// Mitsubishi GX Works2 project: BookEX6_33 Bit   PLC: Q13UDV

// global labels: Global
VAR_GLOBAL
  bVar0 AT M5000 : BOOL;
  abArray0 AT M5010 : ARRAY [0..49] OF BOOL;
  sStr0 AT D5000 : STRING[199];
  sStr1 AT D5100 : STRING[199];
  sStr2 AT D5200 : STRING[199];
  sStr3 AT D5300 : STRING[199];
  sStr4 AT D5400 : STRING[199];
  sStr5 AT D5500 : STRING[199];
  sStr6 AT D5600 : STRING[199];
  sStr7 AT D5700 : STRING[199];
  sStr8 AT D5800 : STRING[199];
  sStr9 AT D5900 : STRING[199];
  iVar0 AT D4500 : INT;
  iVar1 AT D4501 : INT;
  iVar2 AT D4502 : INT;
  iVar3 AT D4503 : INT;
  iVar4 AT D4504 : INT;
  iVar5 AT D4505 : INT;
  iVar6 AT D4506 : INT;
  iVar7 AT D4507 : INT;
  iVar8 AT D4508 : INT;
  iVar9 AT D4509 : INT;
  dVar0 AT D4510 : DINT;
  dVar1 AT D4512 : DINT;
  dVar2 AT D4514 : DINT;
  dVar3 AT D4516 : DINT;
  dVar4 AT D4518 : DINT;
  dVar5 AT D4520 : DINT;
  dVar6 AT D4522 : DINT;
  dVar7 AT D4524 : DINT;
  dVar8 AT D4526 : DINT;
  dVar9 AT D4528 : DINT;
  wVar0 AT D4530 : WORD;
  wVar1 AT D4531 : WORD;
  wVar2 AT D4532 : WORD;
  wVar3 AT D4533 : WORD;
  wVar4 AT D4534 : WORD;
  wVar5 AT D4535 : WORD;
  wVar6 AT D4536 : WORD;
  wVar7 AT D4537 : WORD;
  wVar8 AT D4538 : WORD;
  wVar9 AT D4539 : WORD;
  dwVar0 AT D4540 : DWORD;
  dwVar1 AT D4542 : DWORD;
  dwVar2 AT D4544 : DWORD;
  dwVar3 AT D4546 : DWORD;
  dwVar4 AT D4548 : DWORD;
  dwVar5 AT D4550 : DWORD;
  dwVar6 AT D4552 : DWORD;
  dwVar7 AT D4554 : DWORD;
  dwVar8 AT D4556 : DWORD;
  dwVar9 AT D4558 : DWORD;
  fsVar0 AT D4560 : REAL;
  fsVar1 AT D4562 : REAL;
  fsVar2 AT D4564 : REAL;
  fsVar3 AT D4566 : REAL;
  fsVar4 AT D4568 : REAL;
  fsVar5 AT D4570 : REAL;
  fsVar6 AT D4572 : REAL;
  fsVar7 AT D4574 : REAL;
  fsVar8 AT D4576 : REAL;
  fsVar9 AT D4578 : REAL;
  fdVar0 AT D4580 : LREAL;
  tTime0 AT D4620 : TIME;
  tTime1 AT D4622 : TIME;
  tTime2 AT D4624 : TIME;
  tTime3 AT D4626 : TIME;
  tTime4 AT D4628 : TIME;
  tTime5 AT D4630 : TIME;
  tTime6 AT D4632 : TIME;
  tTime7 AT D4634 : TIME;
  tTime8 AT D4636 : TIME;
  tTime9 AT D4638 : TIME;
  tTime10 AT D4640 : TIME;
  bVar1 AT M5001 : BOOL;
  bVar2 AT M5002 : BOOL;
  bVar3 AT M5003 : BOOL;
  bVar4 AT M5004 : BOOL;
  bVar5 AT M5005 : BOOL;
  bVar6 AT M5006 : BOOL;
  bVar7 AT M5007 : BOOL;
  bVar8 AT M5008 : BOOL;
  bVar9 AT M5009 : BOOL;
  abArray1 AT M5060 : ARRAY [0..49] OF BOOL;
  abArray2 AT M5110 : ARRAY [0..49] OF BOOL;
  abArray3 AT M5160 : ARRAY [0..49] OF BOOL;
  abArray4 AT M5210 : ARRAY [0..49] OF BOOL;
  abArray5 AT M5260 : ARRAY [0..49] OF BOOL;
  abArray6 AT M5310 : ARRAY [0..49] OF BOOL;
  abArray7 AT M5360 : ARRAY [0..49] OF BOOL;
  abArray8 AT M5410 : ARRAY [0..49] OF BOOL;
  abArray9 AT M5460 : ARRAY [0..49] OF BOOL;
  fdVar1 AT D4584 : LREAL;
  fdVar2 AT D4588 : LREAL;
  fdVar3 AT D4592 : LREAL;
  fdVar4 AT D4596 : LREAL;
  fdVar5 AT D4600 : LREAL;
  fdVar6 AT D4604 : LREAL;
  fdVar7 AT D4608 : LREAL;
  fdVar8 AT D4612 : LREAL;
  fdVar9 AT D4616 : LREAL;
  afsPen0 AT D2000 : ARRAY [0..499] OF REAL;
  afsPen1 AT D3000 : ARRAY [0..499] OF REAL;
END_VAR
// user libraries (not included): HMI

FUNCTION DBRST
VAR_INPUT
  dw_IN : DWORD;
  i_Pos : INT;
END_VAR
VAR
  dwInput : DWORD;
  dwTmp1 : DWORD;
  dwTmp2 : DWORD;
END_VAR
;
dwTmp1 := H00000001;
dwInput := dw_IN;
DROL(TRUE, i_Pos MOD 32, dwTmp1);
dwTmp2 := dwInput AND NOT dwTmp1;
DBRST := dwTmp2;
END_FUNCTION

FUNCTION DBSET
VAR_INPUT
  dw_IN : DWORD;
END_VAR
VAR
  dwInput : DWORD;
END_VAR
VAR_INPUT
  i_Pos : INT;
END_VAR
VAR
  dwTmp1 : DWORD;
  dwTmp2 : DWORD;
END_VAR
;
dwTmp1 := H00000001;
dwInput := dw_IN;
DROL(TRUE, i_Pos MOD 32, dwTmp1);
dwTmp2 := dwInput OR dwTmp1;
DBSET := dwTmp2;
END_FUNCTION

FUNCTION newDTEST
VAR_INPUT
  dw_IN : DWORD;
  i_Pos : INT;
END_VAR
VAR
  dwInput : DWORD;
  dwTmp1 : DWORD;
  dwTmp2 : DWORD;
END_VAR
;
dwTmp1 := H00000001;
dwInput := dw_IN;
DROL(TRUE, i_Pos MOD 32, dwTmp1);
dwTmp2 := dwInput AND dwTmp1;
newDTEST := dwTmp2 = dwTmp1;
END_FUNCTION

PROGRAM ExBKRST
(* structured ladder/FBD written out as ST: instructions are called as NAME(EN, inputs, outputs); _pN, _eN, _tN stand for wires *)
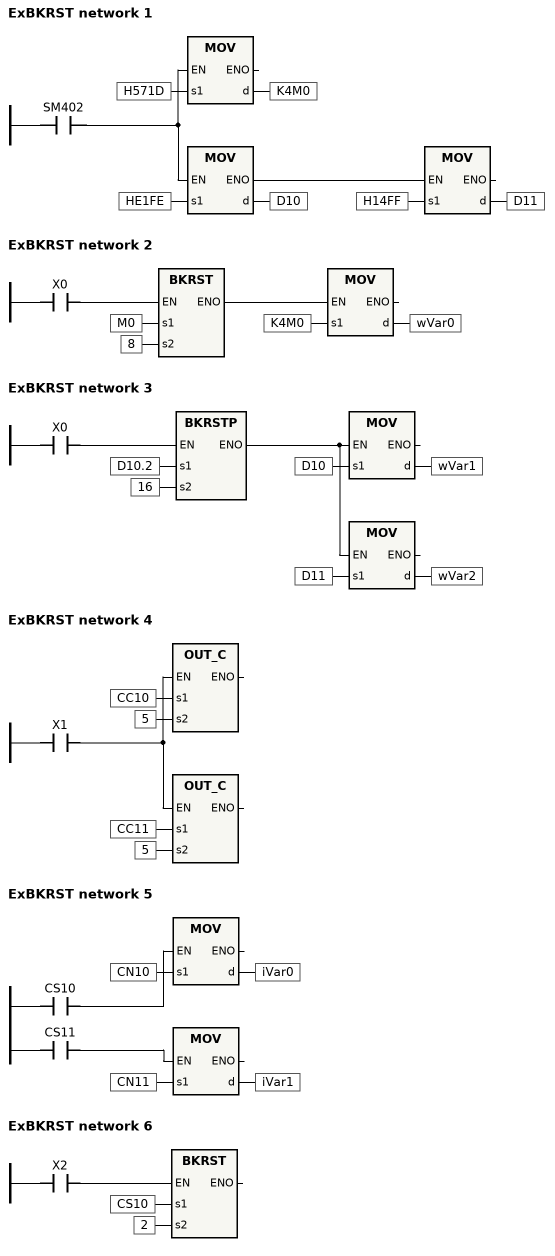
(* network 1 *)
MOV(SM402, H571D, K4M0);
_e1 := MOV(SM402, HE1FE, D10);
MOV(_e1, H14FF, D11);
(* network 2 *)
_e1 := BKRST(X0, M0, 8);
MOV(_e1, K4M0, wVar0);
(* network 3 *)
_e1 := BKRSTP(X0, D10.2, 16);
MOV(_e1, D10, wVar1);
MOV(_e1, D11, wVar2);
(* network 4 *)
OUT_C(X1, CC10, 5);
OUT_C(X1, CC11, 5);
(* network 5 *)
MOV(CS10, CN10, iVar0);
MOV(CS11, CN11, iVar1);
(* network 6 *)
BKRST(X2, CS10, 2);
END_PROGRAM

PROGRAM ExBSET
(* structured ladder/FBD written out as ST: instructions are called as NAME(EN, inputs, outputs); _pN, _eN, _tN stand for wires *)
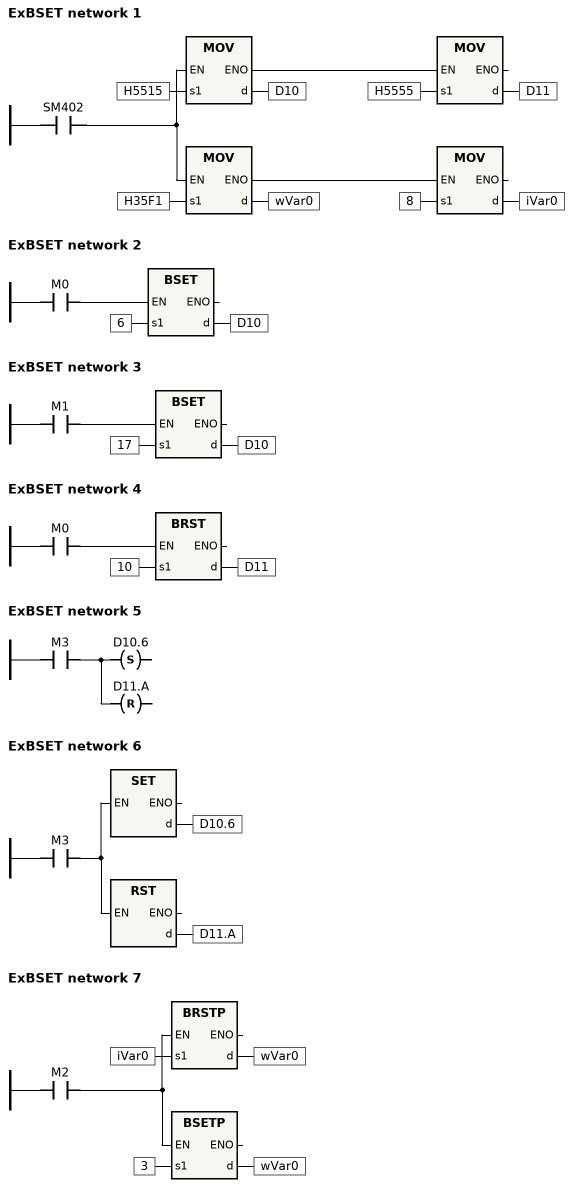
(* network 1 *)
_e1 := MOV(SM402, H5515, D10);
MOV(_e1, H5555, D11);
_e2 := MOV(SM402, H35F1, wVar0);
MOV(_e2, 8, iVar0);
(* network 2 *)
BSET(M0, 6, D10);
(* network 3 *)
BSET(M1, 17, D10);
(* network 4 *)
BRST(M0, 10, D11);
(* network 5 *)
SET(M3, D10.6);
RST(M3, D11.A);
(* network 6 *)
SET(M3, D10.6);
RST(M3, D11.A);
(* network 7 *)
BRSTP(M2, iVar0, wVar0);
BSETP(M2, 3, wVar0);
END_PROGRAM

PROGRAM ExLib
(* structured ladder/FBD written out as ST: instructions are called as NAME(EN, inputs, outputs); _pN, _eN, _tN stand for wires *)
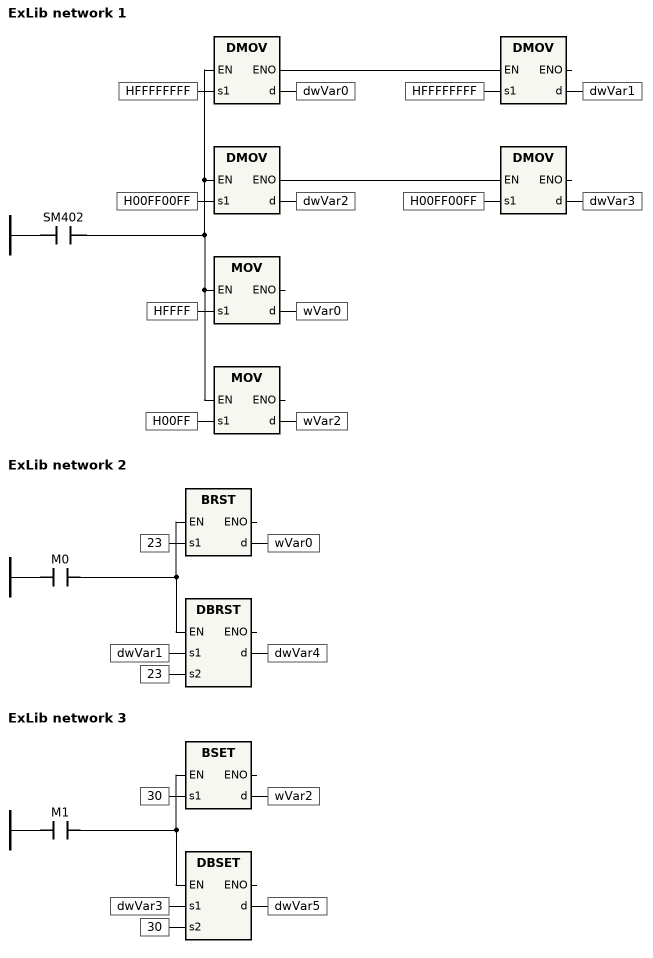
(* network 1 *)
_e1 := DMOV(SM402, HFFFFFFFF, dwVar0);
DMOV(_e1, HFFFFFFFF, dwVar1);
_e2 := DMOV(SM402, H00FF00FF, dwVar2);
DMOV(_e2, H00FF00FF, dwVar3);
MOV(SM402, HFFFF, wVar0);
MOV(SM402, H00FF, wVar2);
(* network 2 *)
BRST(M0, 23, wVar0);
DBRST(M0, dwVar1, 23, dwVar4);
(* network 3 *)
BSET(M1, 30, wVar2);
DBSET(M1, dwVar3, 30, dwVar5);
END_PROGRAM

PROGRAM ExTEST
(* structured ladder/FBD written out as ST: instructions are called as NAME(EN, inputs, outputs); _pN, _eN, _tN stand for wires *)
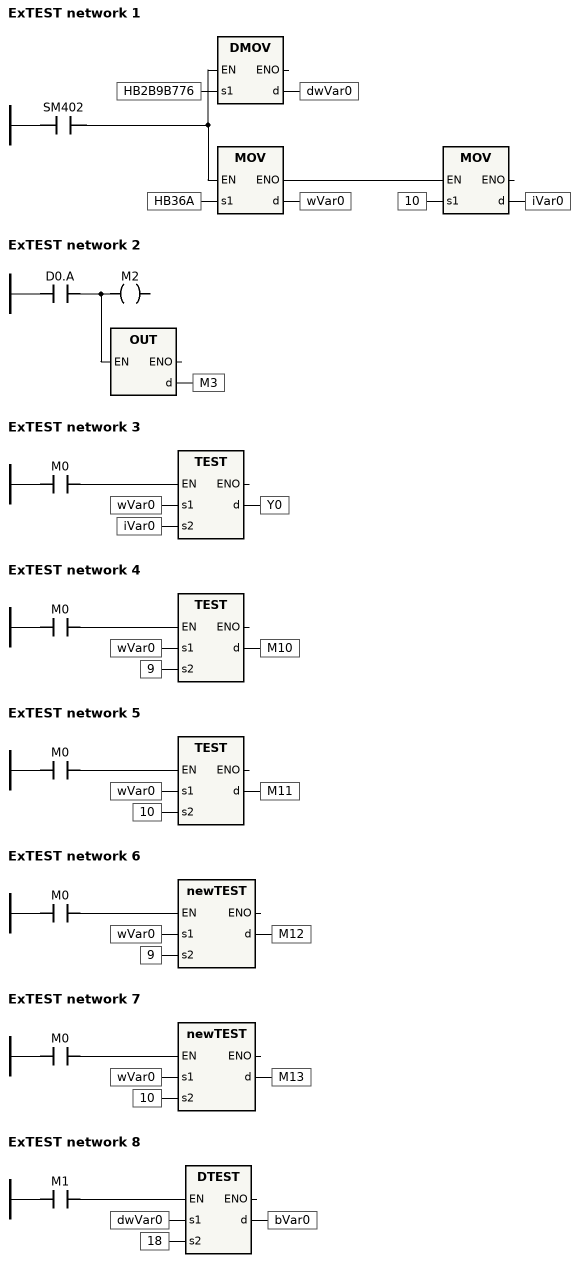
(* network 1 *)
DMOV(SM402, HB2B9B776, dwVar0);
_e1 := MOV(SM402, HB36A, wVar0);
MOV(_e1, 10, iVar0);
(* network 2 *)
M2 := D0.A;
OUT(D0.A, M3);
(* network 3 *)
TEST(M0, wVar0, iVar0, Y0);
(* network 4 *)
TEST(M0, wVar0, 9, M10);
(* network 5 *)
TEST(M0, wVar0, 10, M11);
(* network 6 *)
newTEST(M0, wVar0, 9, M12);
(* network 7 *)
newTEST(M0, wVar0, 10, M13);
(* network 8 *)
DTEST(M1, dwVar0, 18, bVar0);
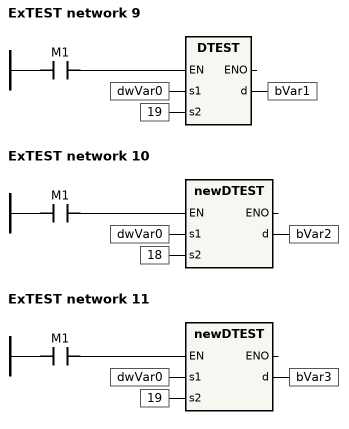
(* network 9 *)
DTEST(M1, dwVar0, 19, bVar1);
(* network 10 *)
newDTEST(M1, dwVar0, 18, bVar2);
(* network 11 *)
newDTEST(M1, dwVar0, 19, bVar3);
END_PROGRAM

FUNCTION newTEST
VAR_INPUT
  w_IN : WORD;
  i_Pos : INT;
END_VAR
VAR
  wInput : WORD;
  wTmp1 : WORD;
  wTmp2 : WORD;
END_VAR
;
wTmp1 := H0001;
wInput := w_IN;
ROL(TRUE, i_Pos MOD 16, wTmp1);
wTmp2 := wInput AND wTmp1;
newTEST := wTmp2 = wTmp1;
END_FUNCTION
